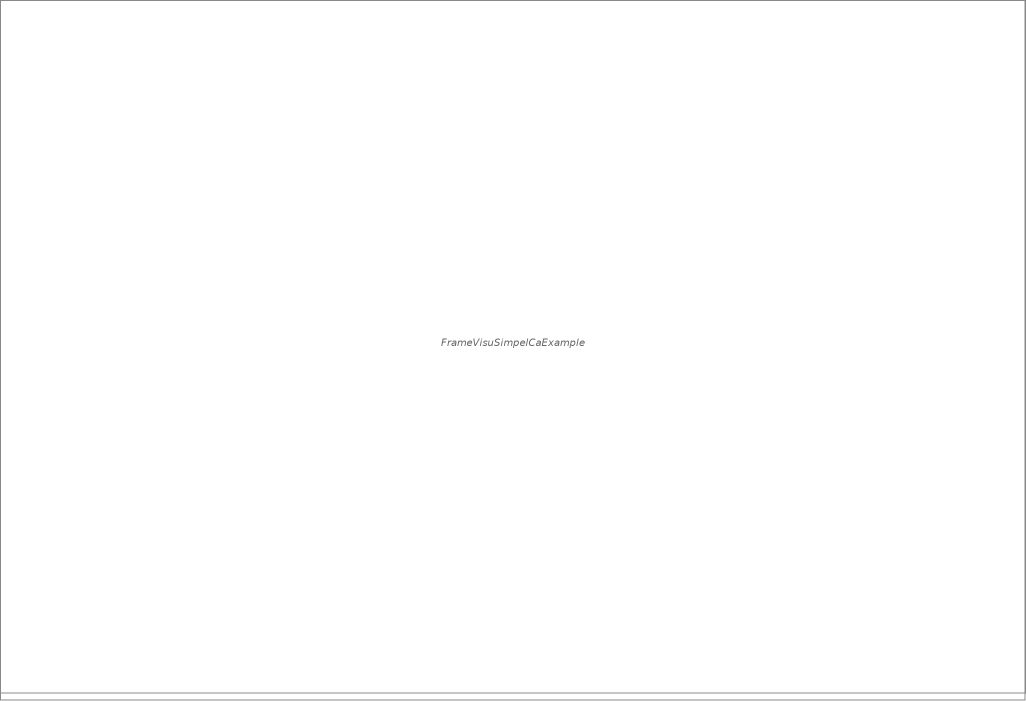
VISUALIZATION CA_Visu  // 1026x701
VAR_IN_OUT
	
END_VAR

VAR
	bShowDisclaimer		: BOOL;
END_VAR
    Frame (0,-8 1026x701)
        shows FrameVisuSimpelCaExample(stVisuIO := MAIN.fbSimpleCaMove.stVisuIO)
END_VISUALIZATION

(* stored: Version 1.1.0.1, ProductVersion 3.1.4024.12
   Visu CA_Visu: Id {a8d2cf77-7820-4de8-84b9-43b6856627bd} *)
